% RSLogix 500 project Pump_ANA_Alarms_Showcase.RSS, saved by version 8.30.00.16 %
PROJECT "UNTITLED"    % processor: Bul.1763 MicroLogix 1100 Series B %

PROGRAM FILES
  LAD 2 "MAIN"  4 rungs
  LAD 3 "ALARMS"  7 rungs
  LAD 4 "ANALOG I/O"  4 rungs
  LAD 5 "CONTROLS"  6 rungs

DATA FILES
  O0 OUTPUT  7 elements
  I1 INPUT  13 elements
  S2 STATUS  66 elements
  B3 BINARY  1 elements
  T4 TIMER  4 elements
  C5 COUNTER  1 elements
  R6 CONTROL  1 elements
  N7 INTEGER  1 elements
  F8 FLOAT  1 elements

LADDER 2 "MAIN"
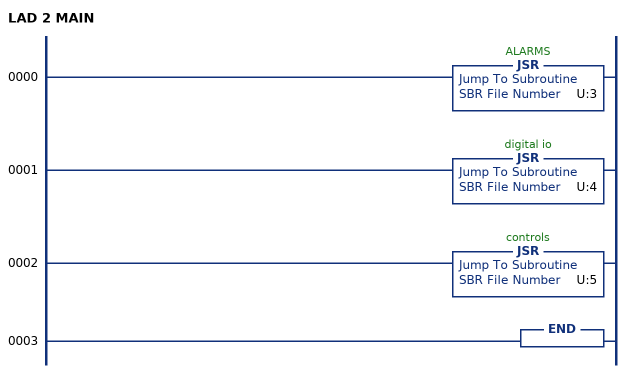
% Rung: 0 %
SOR JSR U:3 EOR
%   U:3  "ALARMS" %
% Rung: 1 %
SOR JSR U:4 EOR
%   U:4  "digital io" %
% Rung: 2 %
SOR JSR U:5 EOR
%   U:5  "controls" %
% Rung: 3 %
SOR END EOR

LADDER 3 "ALARMS"
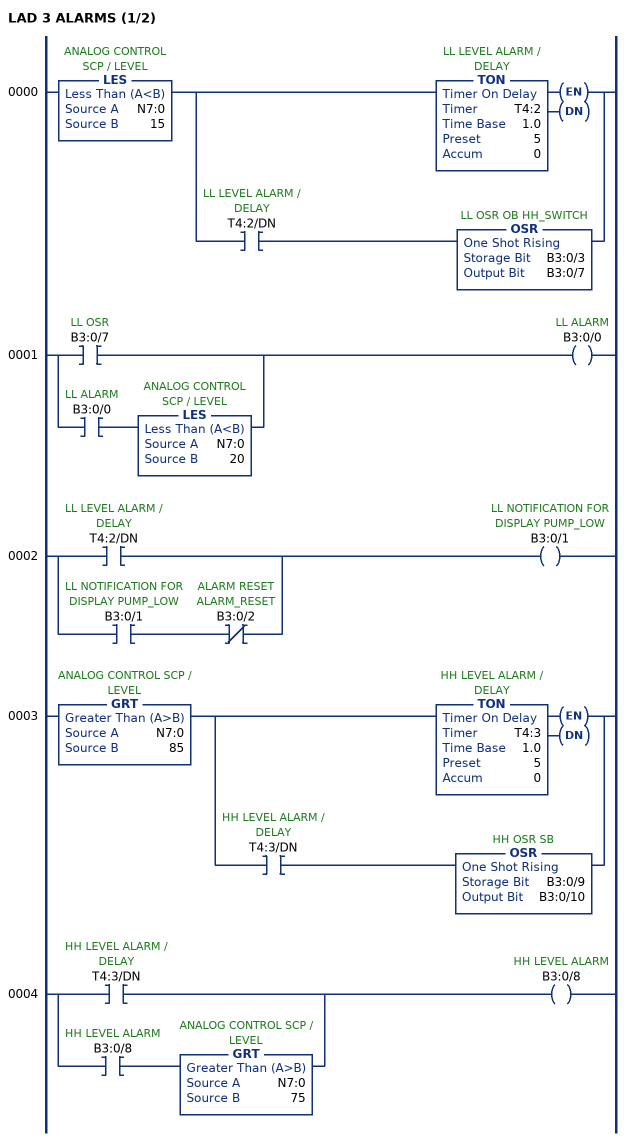
% Rung: 0 %
SOR LES N7:0 15 BST TON T4:2 1.0 5 0 NXB XIC T4:2/DN OSR B3:0/3 B3:0/7 BND EOR
%   N7:0  "ANALOG CONTROL SCP / LEVEL" %
%   T4:2  "LL LEVEL ALARM / DELAY" %
%   B3:0/3  HH_SWITCH  "LL OSR OB" %
%   B3:0/7  "LL OSR" %
% Rung: 1 %
SOR BST XIC B3:0/7 NXB XIC B3:0/0 LES N7:0 20 BND OTE B3:0/0 EOR
%   B3:0/7  "LL OSR" %
%   B3:0/0  "LL ALARM" %
%   N7:0  "ANALOG CONTROL SCP / LEVEL" %
% Rung: 2 %
SOR BST XIC T4:2/DN NXB XIC B3:0/1 XIO B3:0/2 BND OTE B3:0/1 EOR
%   T4:2  "LL LEVEL ALARM / DELAY" %
%   B3:0/1  PUMP_LOW  "LL NOTIFICATION FOR DISPLAY" %
%   B3:0/2  ALARM_RESET  "ALARM RESET" %
% Rung: 3 %
SOR GRT N7:0 85 BST TON T4:3 1.0 5 0 NXB XIC T4:3/DN OSR B3:0/9 B3:0/10 BND EOR
%   N7:0  "ANALOG CONTROL SCP / LEVEL" %
%   T4:3  "HH LEVEL ALARM / DELAY" %
%   B3:0/9  "HH OSR SB" %
%   B3:0/10  "HH OUTPUT BIT" %
% Rung: 4 %
SOR BST XIC T4:3/DN NXB XIC B3:0/8 GRT N7:0 75 BND OTE B3:0/8 EOR
%   T4:3  "HH LEVEL ALARM / DELAY" %
%   B3:0/8  "HH LEVEL ALARM" %
%   N7:0  "ANALOG CONTROL SCP / LEVEL" %

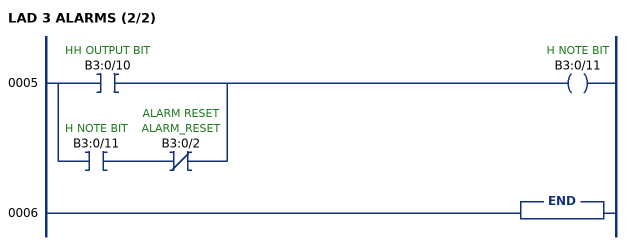
% Rung: 5 %
SOR BST XIC B3:0/10 NXB XIC B3:0/11 XIO B3:0/2 BND OTE B3:0/11 EOR
%   B3:0/10  "HH OUTPUT BIT" %
%   B3:0/11  "H NOTE BIT" %
%   B3:0/2  ALARM_RESET  "ALARM RESET" %
% Rung: 6 %
SOR END EOR

LADDER 4 "ANALOG I/O"
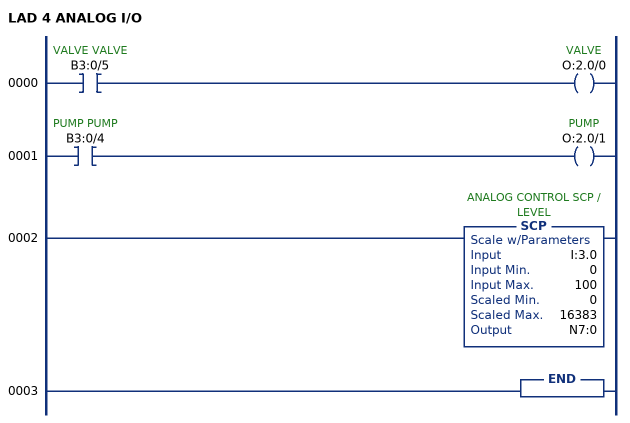
% Rung: 0 %
SOR XIC B3:0/5 OTE O:2.0/0 EOR
%   B3:0/5  VALVE  "VALVE" %
%   O:2.0/0  "VALVE" %
% Rung: 1 %
SOR XIC B3:0/4 OTE O:2.0/1 EOR
%   B3:0/4  PUMP  "PUMP" %
%   O:2.0/1  "PUMP" %
% Rung: 2 %
SOR SCP I:3.0 0 100 0 16383 N7:0 EOR
%   I:3.0  "LEVEL" %
%   N7:0  "ANALOG CONTROL SCP / LEVEL" %
% Rung: 3 %
SOR END EOR

LADDER 5 "CONTROLS"
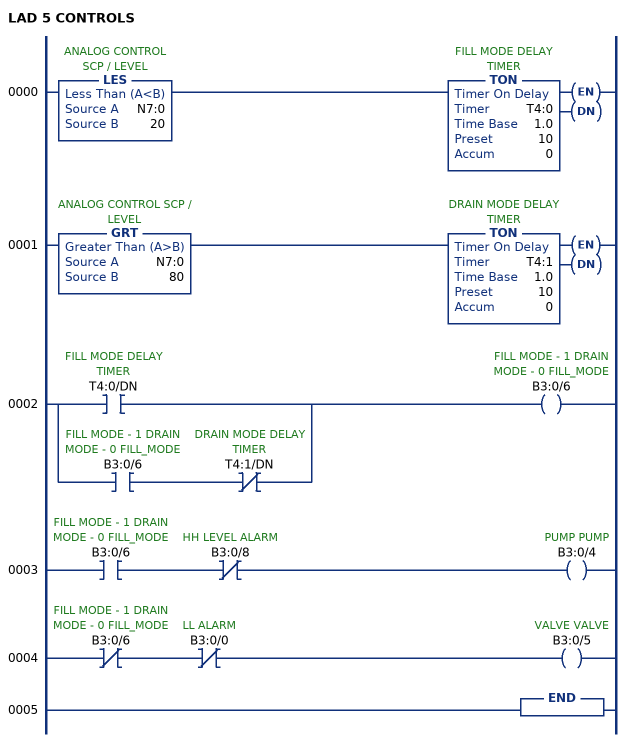
% Rung: 0 %
SOR LES N7:0 20 TON T4:0 1.0 10 0 EOR
%   N7:0  "ANALOG CONTROL SCP / LEVEL" %
%   T4:0  "FILL MODE DELAY TIMER" %
% Rung: 1 %
SOR GRT N7:0 80 TON T4:1 1.0 10 0 EOR
%   N7:0  "ANALOG CONTROL SCP / LEVEL" %
%   T4:1  "DRAIN MODE DELAY TIMER" %
% Rung: 2 %
SOR BST XIC T4:0/DN NXB XIC B3:0/6 XIO T4:1/DN BND OTE B3:0/6 EOR
%   T4:0/DN  "FILL MODE DELAY TIMER" %
%   B3:0/6  FILL_MODE  "FILL MODE - 1 DRAIN MODE - 0" %
%   T4:1  "DRAIN MODE DELAY TIMER" %
% Rung: 3 %
SOR XIC B3:0/6 XIO B3:0/8 OTE B3:0/4 EOR
%   B3:0/6  FILL_MODE  "FILL MODE - 1 DRAIN MODE - 0" %
%   B3:0/8  "HH LEVEL ALARM" %
%   B3:0/4  PUMP  "PUMP" %
% Rung: 4 %
SOR XIO B3:0/6 XIO B3:0/0 OTE B3:0/5 EOR
%   B3:0/6  FILL_MODE  "FILL MODE - 1 DRAIN MODE - 0" %
%   B3:0/0  "LL ALARM" %
%   B3:0/5  VALVE  "VALVE" %
% Rung: 5 %
SOR END EOR

OTHER DOCUMENTED ADDRESSES
  B4:1  "test"
  I:1.0/0  "LL switch input"
  I:1.0/1  "L switch input"
  I:1.0/2  "H INPUT"
  I:1.0/3  "HH INPUT"
  I:3.0/0  "1"
  O:0  "VALVE"
  O:1  "PUMP"

REVISION NOTES
  0: Beta v.1
  1: Final 1.0
  2: v3.1

DATA TABLE (non-zero values as saved)
DATA T4
% .PRE .ACC %
% T4:0 % 10 0
% T4:1 % 10 0
% T4:2 % 5 0
% T4:3 % 5 0
